PROGRAM errorShutdown
VAR
END_VAR

//Set all of the lights to false
Glbl.northStraightActive := FALSE;
Glbl.northLeftActive := FALSE;
Glbl.southStraightActive := FALSE;
Glbl.southLeftActive := FALSE;
Glbl.eastStraightActive := FALSE;
Glbl.eastLeftActive := FALSE;
Glbl.westStraightActive := FALSE;
Glbl.westLeftActive := FALSE;


//Turn all the lights to red, turn the crosswalks to red, make sure no cars can go until the error is resolved
NorthLight_Control.StraightGreenLight := FALSE;
NorthLight_Control.StraightYellowLight := FALSE;
NorthLight_Control.StraightRedLight := TRUE;
NorthLight_Control.LeftGreenLight := FALSE;
NorthLight_Control.LeftYellowLight := FALSE;
NorthLight_Control.LeftRedLight := TRUE;
NorthLight_Control.CrosswalkLight := FALSE;

SouthLight_Control.StraightGreenLight := FALSE;
SouthLight_Control.StraightYellowLight := FALSE;
SouthLight_Control.StraightRedLight := TRUE;
SouthLight_Control.LeftGreenLight := FALSE;
SouthLight_Control.LeftYellowLight := FALSE;
SouthLight_Control.LeftRedLight := TRUE;
SouthLight_Control.CrosswalkLight := FALSE;

EastLight_Control.StraightGreenLight := FALSE;
EastLight_Control.StraightYellowLight := FALSE;
EastLight_Control.StraightRedLight := TRUE;
EastLight_Control.LeftGreenLight := FALSE;
EastLight_Control.LeftYellowLight := FALSE;
EastLight_Control.LeftRedLight := TRUE;
EastLight_Control.CrosswalkLight := FALSE;

WestLight_Control.StraightGreenLight := FALSE;
WestLight_Control.StraightYellowLight := FALSE;
WestLight_Control.StraightRedLight := TRUE;
WestLight_Control.LeftGreenLight := FALSE;
WestLight_Control.LeftYellowLight := FALSE;
WestLight_Control.LeftRedLight := TRUE;
WestLight_Control.CrosswalkLight := FALSE;

END_PROGRAM

(* stored: Version 1.1.0.1, ProductVersion 3.1.4022.10
   POU errorShutdown: Id {6b47d90c-6e80-48fd-b748-5a86d791bab7}, SpecialFunc None *)
